(* IEC 61131-3 sources: traffic-lights/PLC_TrafficLights/Class/SdiasHubBase, 1 file *)

(* ---- SdiasHubBase.st ---- *)
(*!
<Class
	Name               = "SdiasHubBase"
	Revision           = "1.10"
	RealtimeTask       = "false"
	CyclicTask         = "false"
	BackgroundTask     = "false"
	Sigmatek           = "true"
	OSInterface        = "false"
	HighPriority       = "false"
	Automatic          = "false"
	UpdateMode         = "Prescan"
	IconPath           = ".\Class\Tool.ico"
	SharedCommandTable = "true"
	Objectsize         = "(410,120)">
	<Channels>
		<Server Name="ClassSvr" Visualized="false" Initialize="false" WriteProtected="true" Retentive="false" Comment="Connect a SDIAS Client Class"/>
		<Client Name="SplitterPlace" Required="true" Internal="false" Comment="Place of this Splitter"/>
		<Client Name="ToNextSDIAS" Required="true" Internal="false" Comment="Connect to first server of SDIAS Manager or Client"/>
	</Channels>
	<RevDoku>
		<Owner Company="Sigmatek" Author="RamAnd"/>
		<Dokumentation Revision="1.10" Date="01.08.2013" Author="ObeChr" Company="Sigmatek" Description="Comments for Server / Client"/>
		<Dokumentation Revision="1.0" Date="18.07.2013" Author="RamAnd" Company="Sigmatek" Description="First library version"/>
	</RevDoku>
</Class>
*)
SdiasHubBase : CLASS
  //Servers:
	ClassSvr 	: SvrChCmd_DINT;
  //Clients:
	ToNextSDIAS 	: CltChCmd_t_e_VaranErrors;
	SplitterPlace 	: CltCh_DINT;
  //Variables:
  //Functions:

	FUNCTION VIRTUAL GLOBAL ClassSvr::NewInst
		VAR_INPUT
			pPara 	: ^CmdStruct;
			pResult 	: ^results;
		END_VAR
		VAR_OUTPUT
			ret_code 	: iprStates;
		END_VAR;
  //Tables:
	FUNCTION @STD
		VAR_OUTPUT
			ret_code	: CONFSTATES;
		END_VAR;
	FUNCTION GLOBAL TAB @CT_;
END_CLASS;

FUNCTION VIRTUAL GLOBAL SdiasHubBase::ClassSvr::NewInst
	VAR_INPUT
		pPara 	: ^CmdStruct;
		pResult 	: ^results;
	END_VAR
	VAR_OUTPUT
		ret_code 	: iprStates;
	END_VAR

  // use last parameter for port number
  pPara^.aPara[MAXCMDPARA-1] := SplitterPlace;

	ret_code := ToNextSDIAS.NewInst(pPara, pResult);

END_FUNCTION
